INTERFACE ITestEventHandler EXTENDS IEventHandlerBase

METHOD OnCustomEvent
VAR_INPUT
    EventArgs : IStreamReader;
END_VAR
END_METHOD

END_INTERFACE

(* stored: Version 1.1.0.1, ProductVersion 3.1.4024.4
   Itf ITestEventHandler: Id {5c9f4999-f01f-4959-839d-129089c37d61}
   Method OnCustomEvent: Id {83d06d90-640d-490c-a78c-3e28192ff3d4} *)
